TYPE ST_DigitalOutputIO :
STRUCT
	stOut 	AT%Q* : ST_DigitalOutputOut;
END_STRUCT
END_TYPE

(* stored: Version 1.1.0.1, ProductVersion 3.1.4022.9
   DUT ST_DigitalOutputIO: Id {41c5da23-75ec-4487-b224-83440910fe5a} *)
